# EPICS substitutions: mc05/tpmacApp/pmc/xf16ida-mc05-homing.substitutions
file "home_to_limit_template.pmc"
{

pattern
{ AXIS,   PLC,  SERVO,  TIMER }
{ 1,      8,    701,    5511  }
{ 2,      9,    702,    5512  }
{ 3,      10,   703,    5611  }
{ 4,	  11,   704,    5612  }
}
